FUNCTION_BLOCK FB_SimFiller EXTENDS FB_SimStation
VAR_INPUT
END_VAR
VAR_OUTPUT
END_VAR
VAR
	tmrWork						: TON;
END_VAR

METHOD PROTECTED  DoWork : BOOL
VAR_INPUT
END_VAR
tmrWork(IN:=TRUE, PT:=T#2S);
IF tmrWork.Q THEN
	tmrWork(IN:=FALSE);
	DoWork := TRUE;
END_IF
END_METHOD

METHOD PROTECTED  UpdatePartStatus : PVOID
VAR_INPUT
END_VAR
IF pPartStatus <> 0 THEN
	pPartStatus^.bFillerStatus := TRUE;
END_IF
END_METHOD

END_FUNCTION_BLOCK

(* stored: Version 1.1.0.1, ProductVersion 3.1.4024.12
   POU FB_SimFiller: Id {6295f515-0cbf-4a9e-9a05-3f3e3f3d6db2}, SpecialFunc None
   Method DoWork: Id {a766fc47-36c4-453f-960a-63458e5074e8}
   Method UpdatePartStatus: Id {5b766525-df15-487b-a5df-cb66138f8ea6} *)
